// TIA Portal V16 export
// export: Created 2022-02-04T14:40:23.6506352Z, ExportSetting WithDefaults, DisplayName Totally Integrated Automation Portal, DisplayVersion V16 Update 1, DisplayName TIA Portal Version Control Interface, DisplayVersion V16, DisplayName TIA Portal Openness, DisplayVersion V16, DisplayName SINAMICS Startdrive Advanced, DisplayVersion V16 Update 5, DisplayName SINAMICS Startdrive G130, G150, S120, S150, SINAMICS MV, S210, DisplayVersion V16 Update 5, DisplayName SINAMICS Startdrive G110M, G120, G120C, G120D, G120P, G115D, DisplayVersion V16 Update 5, DisplayName STEP 7 Professional, DisplayVersion V16, DisplayName STEP 7 Safety, DisplayVersion V16, DisplayName WinCC Advanced, DisplayVersion V16, DisplayName SIMATIC Visualization Architect, DisplayVersion V16
DATA_BLOCK "FB_Ramp_DB"   // DB15
VERSION : 0.1
// stored: AutoNumber true, InstanceOfName FB_Ramp, InstanceOfType FB
"FB_Ramp"
   // VAR_INPUT
   //    add_lay : Bool;
   //    to_empty : Bool;
   //    new_packet : Bool;
   //    push_packet : Bool;
   //    pick_gaskets : Bool;
   //    gaskets_acquire : Bool;
   //    gaskets_released : Bool;
   //    gaskets_busy : Bool;
   //    mode_no_gasket : Bool;
   //    forks_start_sensor : Bool;
   //    open_lodems_sensor : Bool;
   //    top_sensor : Bool;
   //    mid_sensor : Bool;
   //    low_sensor : Bool;
   //    QPLanksLayers : Int;
   // END_VAR
   // VAR_OUTPUT
   //    carousel_full_reset : Bool;
   //    last_lay : Bool;
   //    down_working : Bool;
   //    make_gasket_layer : Bool;
   //    ramp_not_up : Bool;
   //    ramp_not_down : Bool;
   //    CMD_On : Bool;
   //    CMD_Mid : Bool;
   //    CMD_Off : Bool;
   //    CMD_OpenLodems : Bool;
   //    CMD_CloseLodems : Bool;
   //    layer_holded : Int;
   // END_VAR
   // VAR RETAIN
   //    s_busy : Bool;
   //    s_lay_cmd_permission : Bool;
   //    _State : Int;
   // END_VAR
BEGIN
END_DATA_BLOCK
